// TIA Portal V18 export
// export: Created 2025-12-01T12:39:35.8550761Z, ExportSetting None, DisplayName Totally Integrated Automation Portal, DisplayVersion V18 Update 5, DisplayName TIA Portal Openness, DisplayVersion V18 Update 5, DisplayName TIA Portal Teamcenter Gateway, DisplayVersion V18, DisplayName TIA Portal Version Control Interface, DisplayVersion V18, DisplayName STEP 7 Professional, DisplayVersion V18 Update 5, DisplayName STEP 7 Safety, DisplayVersion V18, DisplayName WinCC Professional, DisplayVersion V18 Update 5
VAR_GLOBAL   // PLC tag table "Marking"
END_VAR
VAR_GLOBAL CONSTANT   // user constants
   MODE_LASER_MARKING_IDLE : Int := 0;
   MODE_LASER_MARKING_START : Int := 1;
   MODE_LASER_MARKING_WRITE : Int := 2;
   MODE_LASER_MARKING_WRITE_ALL : Int := 3;
   MODE_LASER_MARKING_READ_CODE : Int := 4;
END_VAR
